PROGRAM AxisStatusDataStore
VAR
	idx				: INT:=1;
	count			: INT:=0;
END_VAR

FOR idx:=1 TO No DO
	RingBufferAxesPosBuf[idx].SetPos[count] := Axis[Idx].Axis.NcToPlc.SetPos;
	RingBufferAxesPosBuf[idx].ActPos[count] := Axis[Idx].Axis.NcToPlc.ActPos;
	RingBufferAxesVelBuf[idx].SetVel[count] := Axis[Idx].Axis.NcToPlc.SetVelo;
	RingBufferAxesVelBuf[idx].ActVel[count] := Axis[Idx].Axis.NcToPlc.ActVelo;
	RingBufferAxesTrqBuf[idx].Trq[count] := AxesTorque[Idx];
END_FOR

IF count = 999 THEN
	count := 0;
ELSE
	count := count + 1;
END_IF

END_PROGRAM

(* stored: Version 1.1.0.1, ProductVersion 3.1.4024.9
   POU AxisStatusDataStore: Id {9d47c4a0-46c5-48a4-acdc-42bb4c87d2ef}, SpecialFunc None *)
